PROGRAM LOAD_FUKUDA
VAR_INPUT

END_VAR

VAR
	TMR_DELAY: TON;
	TMR1:TON;
	TMR_STOPPER_A: TON;
	TMR_STOPPER_B: TON;
	I_FUKUDA_TRANSFER_AT_BACK_BTHEN: INT;
	TMR_ALARM: TON;
END_VAR

IF 	INPUT_VAR.TRANSPORT_IDX=0 AND 	INPUT_VAR.STATION_LOAD_IDX=0 AND 	INPUT_VAR.JIG_LOAD_IDX =0 THEN
	INPUT_VAR.TRANSPORT_IDX:=	INPUT_VAR.I_CURRENT_TRANSACTION.TRANSPORT_INDEX;
	INPUT_VAR.STATION_LOAD_IDX:=INPUT_VAR.I_CURRENT_TRANSACTION.STATION_NUMBER_LOAD;
	INPUT_VAR.JIG_LOAD_IDX :=	INPUT_VAR.I_CURRENT_TRANSACTION.JIG_INDEX_LOAD;
ELSE
CASE INPUT_VAR.I_CASE OF
0: //standby near lotbox
	IF INPUT_VAR.ACTIVE_ID=6 THEN
		INPUT_VAR.ACTIVE_ID:=1;
	END_IF
	
	INPUT_VAR.TRANSPORT_IDX:=	INPUT_VAR.I_CURRENT_TRANSACTION.TRANSPORT_INDEX;
	INPUT_VAR.STATION_LOAD_IDX:=INPUT_VAR.I_CURRENT_TRANSACTION.STATION_NUMBER_LOAD;
	INPUT_VAR.JIG_LOAD_IDX :=	INPUT_VAR.I_CURRENT_TRANSACTION.JIG_INDEX_LOAD;
	CASE INPUT_VAR.TRANSPORT_IDX OF
		2 : FUKUDA_MOVE(STEP_DATA_1:=INPUT_VAR.STATION_LOAD_IDX,
				STEP_DATA_2:=3,
				STEP_DATA_3:=INPUT_VAR.JIG_LOAD_IDX,
				STEP_DATA_4:=0,
				STEP_DATA_5:=1);
				INPUT_VAR.O_STOPPER_TRANSFER_B:=FALSE;
		1 : FUKUDA_MOVE(STEP_DATA_1:=INPUT_VAR.STATION_LOAD_IDX,
				STEP_DATA_2:=3,
				STEP_DATA_3:=INPUT_VAR.JIG_LOAD_IDX,
				STEP_DATA_4:=1,
				STEP_DATA_5:=0);
				INPUT_VAR.O_STOPPER_TRANSFER_A:=FALSE;
	END_CASE			
	input_var.O_VACUUM_On:=FALSE;
	input_var.O_VACUUM_OFF:=FALSE;	
			
1: //standby near lotbox
	
	IF INPUT_VAR.ACTIVE_ID=6 THEN
		INPUT_VAR.ACTIVE_ID:=1;
	END_IF
		FUKUDA_MOVE(STEP_DATA_1:=INPUT_VAR.STATION_LOAD_IDX,
				STEP_DATA_2:=4,
				STEP_DATA_3:=INPUT_VAR.JIG_LOAD_IDX,
				STEP_DATA_4:=0,
				STEP_DATA_5:=0);

		CASE INPUT_VAR.TRANSPORT_IDX OF
		1:
			INPUT_VAR.I_LOADING_DONE_A:=FALSE;
		
		2:
			INPUT_VAR.I_LOADING_DONE_B:=FALSE;
	END_CASE
	
				
2://vacuum position 
	IF INPUT_VAR.ACTIVE_ID=6 THEN
		INPUT_VAR.ACTIVE_ID:=1;
	END_IF
	INPUT_VAR.I_CASE:=INPUT_VAR.I_CASE+1;
	(*FUKUDA_MOVE(STEP_DATA_1:=INPUT_VAR.I_CURRENT_TRANSACTION.STATION_NUMBER_LOAD,
				STEP_DATA_2:=4,
				STEP_DATA_3:=INPUT_VAR.I_CURRENT_TRANSACTION.JIG_INDEX_LOAD,
				STEP_DATA_4:=0,
				STEP_DATA_5:=0);
	IF INPUT_VAR.ACTIVE_ID=3 THEN
		input_var.O_VACUUM_ON:=TRUE;
		input_var.O_VACUUM_OFF:=FALSE;	
	END_IF
	*)

3://vacuum position 
	IF INPUT_VAR.ACTIVE_ID=6 THEN
		INPUT_VAR.ACTIVE_ID:=1; 
	END_IF
	//INPUT_VAR.I_CASE:=INPUT_VAR.I_CASE+1;
	//IF INPUT_VAR.O_VACUUM_ON THEN
		FUKUDA_MOVE(STEP_DATA_1:=INPUT_VAR.STATION_LOAD_IDX,
				STEP_DATA_2:=4,
				STEP_DATA_3:=INPUT_VAR.JIG_LOAD_IDX,
				STEP_DATA_4:=0,
				STEP_DATA_5:=0);
	//ELSE
		
	//END_IF
4://vacuum position 
	IF INPUT_VAR.ACTIVE_ID=6 THEN
		INPUT_VAR.ACTIVE_ID:=1;
	END_IF
	input_var.O_VACUUM_ON:=TRUE; 
	input_var.O_VACUUM_OFF:=FALSE;
	 
	//CHECK JIG FUKUDA PRESENCE			
	IF  input_var.O_VACUUM_ON THEN
		TMR1(IN:=INPUT_VAR.I_VACUUM_ON,PT:=T#3S);
	END_IF
	IF TMR1.Q  AND INPUT_VAR.I_VACUUM_ON THEN
		input_var.O_VACUUM_ON:=FALSE;
		INPUT_VAR.JIG_FUKUDA_PRESENCE :=FALSE;
		INPUT_VAR.I_CASE:=10;
	ELSE
				INPUT_VAR.JIG_FUKUDA_PRESENCE :=TRUE;	
				FUKUDA_MOVE(STEP_DATA_1:=INPUT_VAR.STATION_LOAD_IDX,
				STEP_DATA_2:=2,
				STEP_DATA_3:=INPUT_VAR.JIG_LOAD_IDX,
				STEP_DATA_4:=0,
				STEP_DATA_5:=0);
	END_IF
				
		

5://vacuum position 
	IF INPUT_VAR.ACTIVE_ID=6 THEN
		INPUT_VAR.ACTIVE_ID:=1;
	END_IF
	
	FUKUDA_MOVE(STEP_DATA_1:=8,
				STEP_DATA_2:=2,
				STEP_DATA_3:=INPUT_VAR.JIG_LOAD_IDX,
				STEP_DATA_4:=0,
				STEP_DATA_5:=0);
	
6://gripping position
	IF INPUT_VAR.ACTIVE_ID=6 THEN
		INPUT_VAR.ACTIVE_ID:=1;
	END_IF

	FUKUDA_MOVE(STEP_DATA_1:=INPUT_VAR.TRANSPORT_IDX+4,
				STEP_DATA_2:=2,
				STEP_DATA_3:=12,
				STEP_DATA_4:=0,
				STEP_DATA_5:=0);


7://placing onto fukuda transport
	IF INPUT_VAR.ACTIVE_ID=6 THEN
		INPUT_VAR.ACTIVE_ID:=1;
	END_IF
	FUKUDA_MOVE(STEP_DATA_1:=INPUT_VAR.TRANSPORT_IDX+4,
				STEP_DATA_2:=2,
				STEP_DATA_3:=11,
				STEP_DATA_4:=0,
				STEP_DATA_5:=0);

8://placing onto fukuda transport
	IF INPUT_VAR.ACTIVE_ID=6 THEN
		INPUT_VAR.ACTIVE_ID:=1;
	END_IF
	
	FUKUDA_MOVE(STEP_DATA_1:=INPUT_VAR.TRANSPORT_IDX+4,
				STEP_DATA_2:=2,
				STEP_DATA_3:=11,
				STEP_DATA_4:=0,
				STEP_DATA_5:=0);
	(*IF INPUT_VAR.ACTIVE_ID=3 THEN
		input_var.O_VACUUM_On:=FALSE;
		input_var.O_VACUUM_OFF:=TRUE;	
	END_IF
	*)
	
9://homing
	IF INPUT_VAR.ACTIVE_ID=6 THEN
		INPUT_VAR.ACTIVE_ID:=1;
	END_IF
	IF INPUT_VAR.I_VACUUM_ON THEN
		FUKUDA_MOVE(STEP_DATA_1:=INPUT_VAR.TRANSPORT_IDX+4,
				STEP_DATA_2:=1,
				STEP_DATA_3:=13,//11
				STEP_DATA_4:=0,
				STEP_DATA_5:=0);
	ELSE
		input_var.O_VACUUM_On:=FALSE;
		input_var.O_VACUUM_OFF:=TRUE;
	END_IF	
				
10://pusH fukuda transport
	IF INPUT_VAR.ACTIVE_ID=6 THEN
		INPUT_VAR.ACTIVE_ID:=1;
	END_IF
	input_var.O_VACUUM_On:=FALSE;
	input_var.O_VACUUM_OFF:=TRUE;
	CASE INPUT_VAR.TRANSPORT_IDX OF
		2 :
			//IF NOT INPUT_VAR.I_FUKUDA_TRANSFER_AT_FRONT_B   THEN
				FUKUDA_MOVE(STEP_DATA_1:=0,
				STEP_DATA_2:=0,
				STEP_DATA_3:=0,
				STEP_DATA_4:=0,
				STEP_DATA_5:=2);
			//END_IF
				 
		1 : 
			//IF NOT INPUT_VAR.I_FUKUDA_TRANSFER_AT_FRONT_A  THEN
				FUKUDA_MOVE(STEP_DATA_1:=0,
				STEP_DATA_2:=0,
				STEP_DATA_3:=0,
				STEP_DATA_4:=2,
				STEP_DATA_5:=0);
			//END_IF
	END_CASE			 
11:
		input_var.O_VACUUM_On:=FALSE;
		input_var.O_VACUUM_OFF:=FALSE;
		CASE INPUT_VAR.TRANSPORT_IDX OF
		1:	
			TMR_ALARM(IN:= NOT INPUT_VAR.I_FUKUDA_TRANSFER_AT_FRONT_A,PT:=T#50S);
			IF INPUT_VAR.I_FUKUDA_TRANSFER_AT_FRONT_A THEN
				TMR_STOPPER_A(IN:=TRUE,PT:=T#0.8S);
				IF TMR_STOPPER_A.Q THEN 
					TMR_ALARM(IN:=FALSE);
					INPUT_VAR.O_STOPPER_TRANSFER_A:=TRUE;
					INPUT_VAR.I_LOADING_DONE_A:=TRUE;
					TMR1(IN:=FALSE);
					TMR_DELAY(IN:=FALSE);
					input_var.O_VACUUM_On:=FALSE;
					input_var.O_VACUUM_OFF:=TRUE;
					FLAG_VAR.ALLOW_EXECUTE_LOAD_FUKUDA:=FALSE;
					INPUT_G6_VAR.I_G6_ENABLE:=TRUE;
					INPUT_VAR.I_CASE:=100;
				END_IF
				
			ELSE
				TMR_STOPPER_A(IN:=FALSE);
				FUKUDA_MOVE(STEP_DATA_1:=0,
				STEP_DATA_2:=0,
				STEP_DATA_3:=0,
				STEP_DATA_4:=2,
				STEP_DATA_5:=0);
			END_IF 
			
			2:
				TMR_ALARM(IN:= NOT INPUT_VAR.I_FUKUDA_TRANSFER_AT_FRONT_B,PT:=T#50S);
			IF INPUT_VAR.I_FUKUDA_TRANSFER_AT_FRONT_B THEN
				
				TMR_STOPPER_B(IN:=TRUE,PT:=T#0.8S);
				IF TMR_STOPPER_B.Q THEN
					TMR_ALARM(IN:=FALSE);
					INPUT_VAR.O_STOPPER_TRANSFER_B:=TRUE;	
					INPUT_VAR.I_LOADING_DONE_B:=TRUE;
					TMR1(IN:=FALSE);
					TMR_DELAY(IN:=FALSE);
					input_var.O_VACUUM_On:=FALSE;
					input_var.O_VACUUM_OFF:=TRUE;
					FLAG_VAR.ALLOW_EXECUTE_LOAD_FUKUDA:=FALSE;
					INPUT_G6_VAR.I_G6_ENABLE:=TRUE;
					INPUT_VAR.I_CASE:=100;
				END_IF
			ELSE
				TMR_STOPPER_B(IN:=FALSE);
				FUKUDA_MOVE(STEP_DATA_1:=0,
				STEP_DATA_2:=0,
				STEP_DATA_3:=0,
				STEP_DATA_4:=0,
				STEP_DATA_5:=2);
			END_IF
			
	END_CASE 
	IF TMR_ALARM.Q THEN
					INPUT_VAR.I_LOADING_DONE_B:=FALSE;
					TMR1(IN:=FALSE);
					TMR_DELAY(IN:=FALSE);
					input_var.O_VACUUM_On:=FALSE;
					input_var.O_VACUUM_OFF:=FALSE;
					FLAG_VAR.ALLOW_EXECUTE_LOAD_FUKUDA:=FALSE;
					INPUT_VAR.I_CASE:=100;
	END_IF
100:
	
	FLAG_VAR.ALLOW_EXECUTE_LOAD_FUKUDA:=FALSE;								
								
END_CASE 
END_IF

END_PROGRAM

(* stored: Version 1.1.0.1, ProductVersion 3.1.4020.12
   POU LOAD_FUKUDA: Id {4ece86f8-7a37-4f62-b8e7-f3ac9027245d}, SpecialFunc None *)
